// TIA Portal V21 export
DATA_BLOCK "new"   // DB260
{ S7_Optimized_Access := 'FALSE' }
   VAR RETAIN
      "std end press" : String[80] := '$L$REND PRESSURE (BAR)                    :               ';
      "STD STERILE HOLD TEMP" : Array[0..12] of Real;
      "STD STERILE HOLD TIME" : Array[0..12] of Int;
      "STD BAND" : Array[0..12] of Real;
      "STD OVER TEMP" : Array[0..12] of Real;
      "STD ABORT TEMP" : Array[0..12] of Real;
      "STD STERILE STOP TEMP" : Array[0..12] of Real;
      "EXTRA TEMP" : Real := 0.3;
      "HPHV SET TEMP" : Array[0..3] of Real;
      "BOW SET TEMP" : Array[0..3] of Real;
      "HPHV SET TIME" : Array[0..3] of Int;
      "BOW SET TIME" : Array[0..3] of Int;
      "HPHV STOP TEMP" : Real := 120.9;
      "BOW STOP TEMP" : Real := 120.9;
      "JACKET ALARM TIME" : Int := 10;
      "HEATUP ALARM TIME" : Int := 10;
      "TEMP OFFSET" : Array[0..10] of Real;
      "SET VACUUM ALARM TIME" : Int := 30;
      "SET LEAK VCC" : Real := -0.7;
      "SET VCC PRESS" : Real := -0.05;
      "SET DELAY BEFORE HOLD TIME" : Int := 0;
      "SET VCC HOLD TIME" : Int := 10;
      "SET ACCEPTANCE LEAK" : Real := 0.013;
   END_VAR
BEGIN
   "STD STERILE HOLD TEMP"[0..2] := 121.4;
   "STD STERILE HOLD TEMP"[3..5] := 115.0;
   "STD STERILE HOLD TEMP"[6] := 110.0;
   "STD STERILE HOLD TEMP"[7..8] := 100.0;
   "STD STERILE HOLD TEMP"[9..12] := 0.0;
   "STD STERILE HOLD TIME"[0] := 30;
   "STD STERILE HOLD TIME"[1] := 20;
   "STD STERILE HOLD TIME"[2] := 15;
   "STD STERILE HOLD TIME"[3] := 35;
   "STD STERILE HOLD TIME"[4] := 30;
   "STD STERILE HOLD TIME"[5..6] := 15;
   "STD STERILE HOLD TIME"[7] := 35;
   "STD STERILE HOLD TIME"[8] := 20;
   "STD STERILE HOLD TIME"[9..12] := 0;
   "STD BAND"[0..12] := 0.0;
   "STD OVER TEMP"[0..2] := 124.0;
   "STD OVER TEMP"[3..5] := 118.0;
   "STD OVER TEMP"[6] := 113.0;
   "STD OVER TEMP"[7..8] := 103.0;
   "STD OVER TEMP"[9..10] := 124.0;
   "STD OVER TEMP"[11..12] := 0.0;
   "STD ABORT TEMP"[0..2] := 120.5;
   "STD ABORT TEMP"[3..5] := 114.5;
   "STD ABORT TEMP"[6..7] := 109.5;
   "STD ABORT TEMP"[8] := 99.5;
   "STD ABORT TEMP"[9..10] := 120.5;
   "STD ABORT TEMP"[11..12] := 0.0;
   "STD STERILE STOP TEMP"[0..2] := 120.9;
   "STD STERILE STOP TEMP"[3..5] := 114.9;
   "STD STERILE STOP TEMP"[6] := 109.9;
   "STD STERILE STOP TEMP"[7..8] := 99.9;
   "STD STERILE STOP TEMP"[9..12] := 0.0;
   "HPHV SET TEMP"[0] := 114.0;
   "HPHV SET TEMP"[1] := 116.0;
   "HPHV SET TEMP"[2] := 119.0;
   "HPHV SET TEMP"[3] := 0.0;
   "BOW SET TEMP"[0] := 114.0;
   "BOW SET TEMP"[1] := 116.0;
   "BOW SET TEMP"[2] := 119.0;
   "BOW SET TEMP"[3] := 0.0;
   "HPHV SET TIME"[0] := 5;
   "HPHV SET TIME"[1] := 3;
   "HPHV SET TIME"[2] := 2;
   "HPHV SET TIME"[3] := 1;
   "BOW SET TIME"[0] := 5;
   "BOW SET TIME"[1] := 3;
   "BOW SET TIME"[2] := 2;
   "BOW SET TIME"[3] := 0;
   "TEMP OFFSET"[0..1] := 0.0;
   "TEMP OFFSET"[2..3] := 0.2;
   "TEMP OFFSET"[4] := 0.0;
   "TEMP OFFSET"[5] := 0.1;
   "TEMP OFFSET"[6..10] := 0.0;
END_DATA_BLOCK
